FUNCTION_BLOCK Test
VAR
	_process:TestProcess;
	_start, _stop, _running:BOOL;
END_VAR

IF _start THEN
	_process.Start();
	_start := FALSE;
END_IF
IF _stop THEN
	_process.Stop();
	_stop := FALSE;
END_IF
_process();
_running := _process.Running;

END_FUNCTION_BLOCK

(* stored: Version 1.1.0.1, ProductVersion 3.1.4024.2
   POU Test: Id {b3e6b4c9-6024-4350-9951-b167e5227189}, SpecialFunc None *)
